(* IEC 61131-3 sources: CodesysTest/alpha/export/Device.dev/Plc Logic/Application/FBs/Temp Sensors/FB_TemperatureSensor.pou, 1 file *)

(* ---- FB_TemperatureSensor.pou.st ---- *)
(*#-#-#-#-#-#-#-#-#-#---Declaration---#-#-#-#-#-#-#-#-#-#-#-#-#*)

FUNCTION_BLOCK FB_TemperatureSensor IMPLEMENTS ITempSensor
VAR_INPUT
END_VAR
VAR_OUTPUT
END_VAR
VAR
	_instanceName : STRING;			// Instance Name
	_rawTemperatureReading : INT;   // Raw reading from sensor
	_temperatureReadingC : REAL;	// Scaled temperaure reading in degC
	_temperatureReadingF : REAL;	// Scaled temperaure reading in degF
END_VAR
(*#-#-#-#-#-#-#-#-#-#---Implementation---#-#-#-#-#-#-#-#-#-#-#-#-#*)
